// TIA Portal project "FactoryIO_Template_S7-1500_V15_parcial1_terminado" (V15)

(* hardware
DEVICE "S71500/ET200MP-Station_1"  S7-1500 station
   slot 0: "Profilschiene_0"  6ES7 590-1***0-0AA0
   slot 1: "PLC_1"  CPU 1511-1 PN  6ES7 511-1AK00-0AB0  V1.8
   slot 2: "AI 8xU/I/RTD/TC ST_1"  AI 8xU/I/RTD/TC ST  6ES7 531-7KF00-0AB0  V2.0
   slot 3: "AI 8xU/I/RTD/TC ST_2"  AI 8xU/I/RTD/TC ST  6ES7 531-7KF00-0AB0  V2.0
   slot 4: "AI 8xU/I/RTD/TC ST_3"  AI 8xU/I/RTD/TC ST  6ES7 531-7KF00-0AB0  V2.0
   slot 5: "AI 8xU/I/RTD/TC ST_4"  AI 8xU/I/RTD/TC ST  6ES7 531-7KF00-0AB0  V2.0
   slot 6: "DI 16x24VDC BA_1"  DI 16x24VDC BA  6ES7 521-1BH10-0AA0  V1.0
*)

// ===== PLC "PLC_1"  CPU 1511-1 PN =====

VAR_GLOBAL   // PLC tag table "Standard-Variablentabelle"
   "Box_feeder" AT %Q0.0 : Bool;
   "Load_belt" AT %Q0.1 : Bool;
   "Start" AT %I0.0 : Bool;
   "Stop" AT %I0.1 : Bool;
   "Reset" AT %I0.2 : Bool;
   "Manual" AT %I0.3 : Bool;
   "Emergency_stop" AT %I0.5 : Bool;
   "Box_entry" AT %I0.6 : Bool;
   "Turn" AT %Q0.2 : Bool;
   "Pusher_limit" AT %I0.7 : Bool;
   "Push" AT %Q0.3 : Bool;
   "Open_Plate" AT %Q0.4 : Bool;
   "Plate_limit" AT %I1.0 : Bool;
   "Clamp" AT %Q0.5 : Bool;
   "Clamped" AT %I1.1 : Bool;
   "Pallet_feeder" AT %Q0.6 : Bool;
   "Pallet_at_entry" AT %I1.2 : Bool;
   "S1_Elevator_base" AT %I1.3 : Bool;
   "S2_Elevator_base" AT %I1.4 : Bool;
   "Pallet_at_exit" AT %I1.5 : Bool;
   "Exit_conveyor" AT %Q0.7 : Bool;
   "Elevator_moving" AT %I1.6 : Bool;
   "Move_to_limit" AT %Q1.0 : Bool;
   "Elevator_up" AT %Q1.1 : Bool;
   "Warning light" AT %Q1.3 : Bool;
   "Auto" AT %I0.4 : Bool;
   "Elevator_down" AT %Q1.2 : Bool;
   "Contador1" AT %MW10 : Word;
   "Contador2" AT %MW12 : Word;
   "Contador3" AT %MW14 : Word;
   "Contador4" AT %MW16 : Word;
   "Contador5" AT %MW18 : Word;
   "LimiteContador1" AT %MW20 : Word;
   "LimiteContador2" AT %MW22 : Word;
   "Pallet_in_acensor" AT %M100.0 : Bool;
   "Load_pallet" AT %Q1.4 : Bool;
   "Run_machine" AT %M0.0 : Bool;
   "Elevator_Listo_a_cargar" AT %M100.1 : Bool;
   "LimiteContador3" AT %MW24 : Word;
   "Plaforma_llena" AT %M100.2 : Bool;
END_VAR

DATA_BLOCK "GRAPH1_DB"   // DB1
{ S7_Optimized_Access := 'TRUE' }
VERSION : 0.1
// stored: InstanceOfName GRAPH1
"GRAPH1"
BEGIN
END_DATA_BLOCK

DATA_BLOCK "GRAPH2_DB"   // DB2
{ S7_Optimized_Access := 'TRUE' }
VERSION : 0.1
// stored: InstanceOfName GRAPH2
"GRAPH2"
BEGIN
END_DATA_BLOCK

FUNCTION_BLOCK "GRAPH1"   // FB1, GRAPH_PLUS
{ S7_Optimized_Access := 'TRUE' }
VERSION : 0.1
   VAR_INPUT
      OFF_SQ : Bool := false;   // Turn sequence off
      INIT_SQ : Bool := false;   // Set sequence to initial state
      ACK_EF : Bool := false;   // Acknowledge all errors and faults
      S_PREV : Bool := false;   // Output previous step in parameter S_NO
      S_NEXT : Bool := false;   // Indicate next step in parameter S_NO
      SW_AUTO : Bool := false;   // Automatic mode
      SW_TAP : Bool := false;   // Semiautomatic/switch with transition
      SW_TOP : Bool := false;   // Semiautomatic/ignore transition
      SW_MAN : Bool := false;   // Manual mode
      S_SEL : Int := 0;   // Select step to be output to S_NO
      S_ON : Bool := false;   // Activate step indicated in S_NO
      S_OFF : Bool := false;   // Deactivate step indicated S_NO
      T_PUSH : Bool := false;   // Enable transition to switch in semi automatic mode
   END_VAR
   VAR_OUTPUT
      S_NO : Int := 0;   // Step number
      S_MORE : Bool := false;   // More steps are available and can be shown in S_NO
      S_ACTIVE : Bool := false;   // Step indicated in S_NO is active
      ERR_FLT : Bool := false;   // Interlock or supervision group error
      AUTO_ON : Bool := false;   // Automatic mode is active
      TAP_ON : Bool := false;   // Semiautomatic mode/step with transition enabled
      TOP_ON : Bool := false;   // Semiautomatic mode/ignore transition enabled
      MAN_ON : Bool := false;   // Manual mode is active
   END_VAR
   VAR
      HMI_INFO : Array[0..8] of UInt;
      IF_PAR : G7_IfParPlus_V2;
      RT_DATA : G7_RTDataPlus_V2;   // Internal data area
      Trans1 : G7_TransitionPlus_V2;   // Transition structure
      Trans2 : G7_TransitionPlus_V2;   // Transition structure
      Trans3 : G7_TransitionPlus_V2;   // Transition structure
      Trans4 : G7_TransitionPlus_V2;   // Transition structure
      Trans10 : G7_TransitionPlus_V2;   // Transition structure
      Trans12 : G7_TransitionPlus_V2;   // Transition structure
      Trans13 : G7_TransitionPlus_V2;   // Transition structure
      Trans16 : G7_TransitionPlus_V2;   // Transition structure
      Trans17 : G7_TransitionPlus_V2;   // Transition structure
      Trans18 : G7_TransitionPlus_V2;   // Transition structure
      Trans22 : G7_TransitionPlus_V2;   // Transition structure
      Trans24 : G7_TransitionPlus_V2;   // Transition structure
      Trans25 : G7_TransitionPlus_V2;   // Transition structure
      Trans26 : G7_TransitionPlus_V2;   // Transition structure
      Trans27 : G7_TransitionPlus_V2;   // Transition structure
      Trans28 : G7_TransitionPlus_V2;   // Transition structure
      Reposo : G7_StepPlus_V2;   // Step structure
      Bandas_ON : G7_StepPlus_V2;   // Step structure
      Caja_en_psoicion : G7_StepPlus_V2;   // Step structure
      haciendo_push : G7_StepPlus_V2;   // Step structure
      Saliendo_push : G7_StepPlus_V2;   // Step structure
      Push_afuera_regrese : G7_StepPlus_V2;   // Step structure
      Push_regresando : G7_StepPlus_V2;   // Step structure
      box_hacia_load_belt : G7_StepPlus_V2;   // Step structure
      Avanzando_box_en_load_belt : G7_StepPlus_V2;   // Step structure
      Push_en_inicio : G7_StepPlus_V2;   // Step structure
      "6_cajas_en_plato" : G7_StepPlus_V2;   // Step structure
      Intercambiar_sin_turn : G7_StepPlus_V2;   // Step structure
      Intercambiar_con_turn : G7_StepPlus_V2;   // Step structure
      SINI : Array[0..1] of USInt;
      LSTT : Array[0..15] of USInt;
      ATAJ : Array[0..15] of USInt;
      ATAB : Array[0..15] of USInt;
      PSTT : Array[0..15] of USInt;
      NSTT : Array[0..15] of USInt;
      ASSJ : Array[0..12] of USInt;
      ASSB : Array[0..12] of USInt;
      PTTS : Array[0..12] of USInt;
      NTTS : Array[0..12] of USInt;
      SW_SQTS : Array[0..12] of USInt;
      SWITCH : Array[0..4] of USInt;
      TVX : Array[0..7] of USInt;
      TTX : Array[0..7] of USInt;
      TSX : Array[0..1] of USInt;
      S00X : Array[0..1] of USInt;
      SOFFX : Array[0..1] of USInt;
      SONX : Array[0..1] of USInt;
      SAX : Array[0..1] of USInt;
      SERRX : Array[0..13] of USInt;
      SMX : Array[0..13] of USInt;
      S0X : Array[0..13] of USInt;
      S1X : Array[0..13] of USInt;
      IL_ALARM_INST : Program_Alarm;
      SUP_ALARM_INST : Program_Alarm;
      STEP_TIME_ALARM_INST : Program_Alarm;
      IEC_TIMER_INST : IEC_TIMER;
      TRANSACTION_FLAG : Bool := false;
   END_VAR
   // SINI[0] := 2;
   // LSTT[0] := 255;
   // ATAJ[1] := 1;
   // ATAB[1] := 1;
   // PSTT[1] := 1;
   // NSTT[0] := 1;
   // ASSJ[1] := 1;
   // ASSB[1] := 1;
   // PTTS[0] := 255;
   // NTTS[1] := 1;
   // TVX[0] := 16#1;
   // TTX[0] := 16#1;
   // TSX[0] := 16#1;
   // S00X[0] := 16#1;
   // SOFFX[0] := 16#1;
   // SONX[0] := 16#1;
   // SAX[0] := 16#1;
   // SERRX[0] := 16#1;
   // SMX[0] := 16#1;
   // S0X[0] := 16#1;
   // S1X[0] := 16#1;
   // LSTT[1] := 255;
   // LSTT[2] := 255;
   // LSTT[3] := 255;
   // ATAJ[2] := 2;
   // ATAJ[3] := 3;
   // ATAJ[4] := 4;
   // ATAJ[5] := 5;
   // ATAB[2] := 3;
   // ATAB[3] := 2;
   // ATAB[4] := 4;
   // ATAB[5] := 5;
   // PSTT[2] := 2;
   // PSTT[3] := 2;
   // PSTT[4] := 3;
   // PSTT[5] := 4;
   // NSTT[1] := 2;
   // NSTT[2] := 3;
   // NSTT[3] := 7;
   // ASSJ[2] := 2;
   // ASSJ[3] := 3;
   // ASSJ[4] := 4;
   // ASSB[2] := 2;
   // ASSB[3] := 3;
   // ASSB[4] := 4;
   // PTTS[2] := 1;
   // PTTS[3] := 2;
   // PTTS[4] := 4;
   // NTTS[2] := 2;
   // NTTS[3] := 4;
   // NTTS[4] := 5;
   // SW_SQTS[3] := 1;
   // SW_SQTS[4] := 1;
   // LSTT[5] := 255;
   // NSTT[5] := 5;
   // LSTT[4] := 255;
   // LSTT[6] := 255;
   // LSTT[7] := 255;
   // ATAJ[6] := 6;
   // ATAJ[7] := 7;
   // ATAB[6] := 6;
   // ATAB[7] := 7;
   // PSTT[6] := 5;
   // PSTT[7] := 7;
   // NSTT[4] := 4;
   // NSTT[6] := 6;
   // NSTT[7] := 8;
   // ASSJ[5] := 5;
   // ASSJ[6] := 6;
   // ASSB[5] := 5;
   // ASSB[6] := 6;
   // PTTS[5] := 5;
   // PTTS[6] := 6;
   // NTTS[5] := 6;
   // NTTS[6] := 9;
   // SW_SQTS[5] := 1;
   // SW_SQTS[6] := 1;
   // LSTT[8] := 2;
   // LSTT[9] := 255;
   // LSTT[10] := 255;
   // ATAJ[8] := 8;
   // ATAJ[9] := 9;
   // ATAJ[10] := 10;
   // ATAB[8] := 8;
   // ATAB[9] := 9;
   // ATAB[10] := 15;
   // PSTT[8] := 8;
   // PSTT[9] := 6;
   // PSTT[10] := 9;
   // NSTT[8] := 2;
   // NSTT[9] := 9;
   // NSTT[10] := 10;
   // ASSJ[7] := 7;
   // ASSJ[8] := 8;
   // ASSB[7] := 7;
   // ASSB[8] := 8;
   // PTTS[7] := 3;
   // PTTS[8] := 7;
   // NTTS[7] := 7;
   // NTTS[8] := 8;
   // SW_SQTS[7] := 2;
   // SW_SQTS[8] := 2;
   // ATAB[11] := 12;
   // ATAJ[11] := 11;
   // LSTT[11] := 255;
   // PSTT[11] := 10;
   // NSTT[11] := 12;
   // ASSJ[9] := 9;
   // ASSB[9] := 9;
   // PTTS[9] := 9;
   // NTTS[9] := 10;
   // SW_SQTS[9] := 1;
   // LSTT[12] := 255;
   // LSTT[13] := 2;
   // LSTT[14] := 2;
   // LSTT[15] := 2;
   // ATAJ[12] := 12;
   // ATAJ[13] := 13;
   // ATAJ[14] := 14;
   // ATAJ[15] := 15;
   // ATAB[12] := 11;
   // ATAB[13] := 13;
   // ATAB[14] := 14;
   // ATAB[15] := 10;
   // PSTT[12] := 10;
   // PSTT[13] := 11;
   // PSTT[14] := 12;
   // PSTT[15] := 9;
   // NSTT[12] := 11;
   // NSTT[13] := 2;
   // NSTT[14] := 2;
   // NSTT[15] := 2;
   // ASSJ[10] := 10;
   // ASSJ[11] := 11;
   // ASSJ[12] := 12;
   // ASSB[10] := 10;
   // ASSB[11] := 11;
   // ASSB[12] := 12;
   // PTTS[10] := 10;
   // PTTS[11] := 12;
   // PTTS[12] := 11;
   // NTTS[10] := 12;
   // NTTS[11] := 13;
   // NTTS[12] := 14;
   // SW_SQTS[10] := 3;
   // SW_SQTS[11] := 4;
   // SW_SQTS[12] := 5;
BEGIN
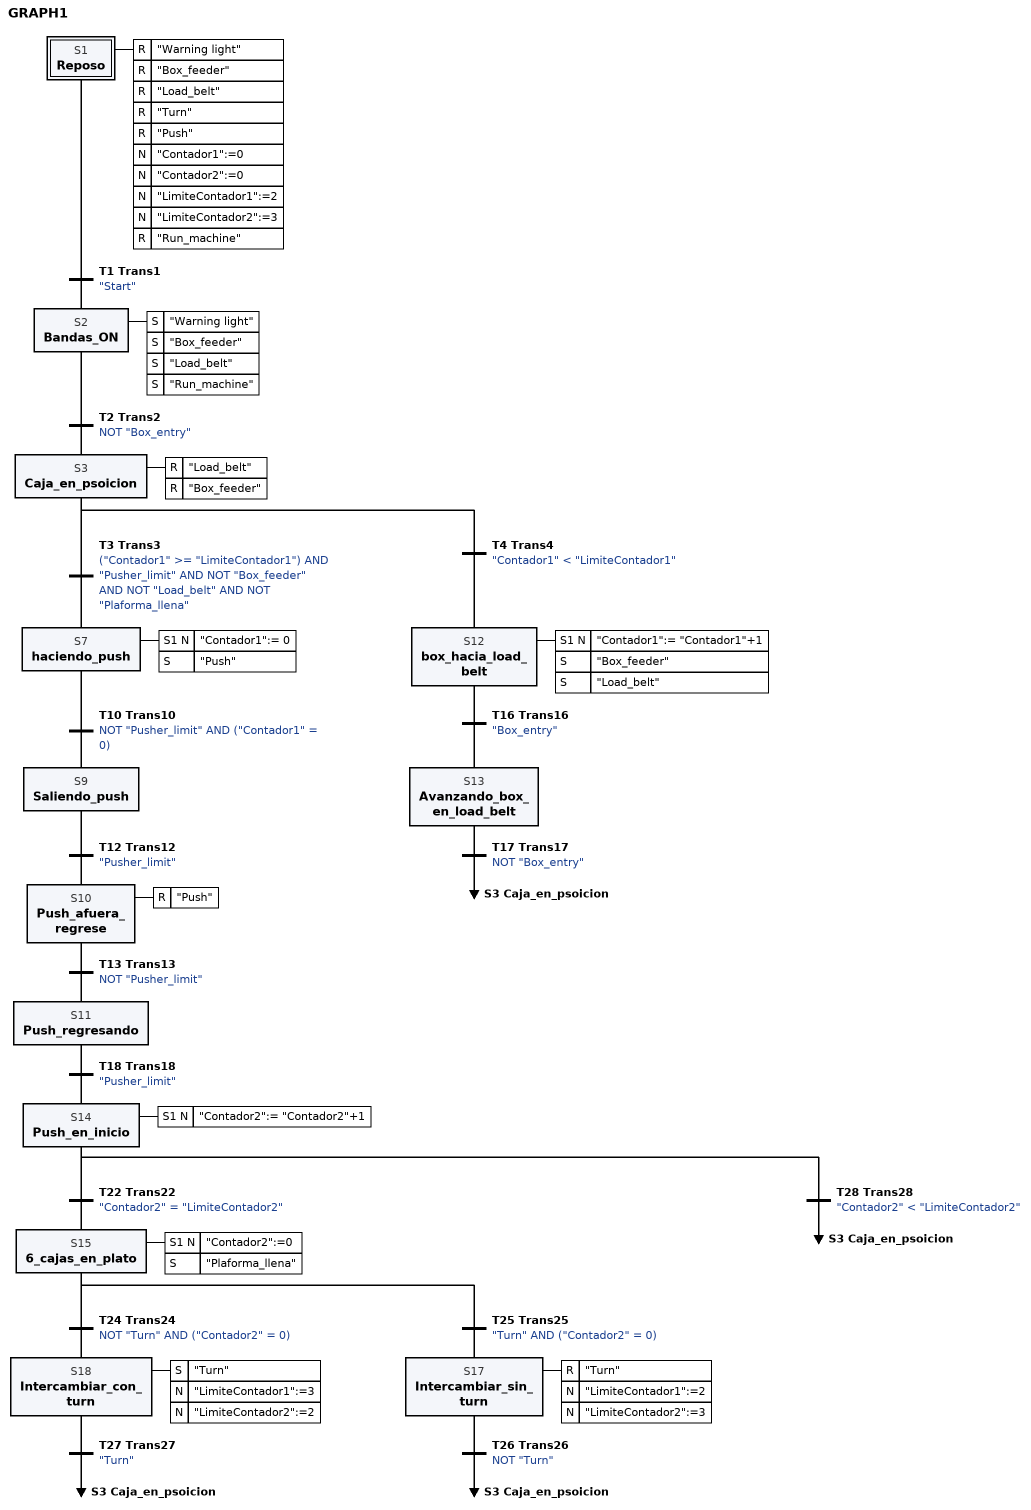
   // sequencer 1
   INITIAL_STEP Reposo:   // S1, max time T#10S, warning time T#7S
              R    "Warning light"
              R    "Box_feeder"
              R    "Load_belt"
              R    "Turn"
              R    "Push"
              N    "Contador1":=0
              N    "Contador2":=0
              N    "LimiteContador1":=2
              N    "LimiteContador2":=3
              R    "Run_machine"
   END_STEP
   TRANSITION Trans1 FROM Reposo TO Bandas_ON   // T1
      := "Start";
   END_TRANSITION
   STEP Bandas_ON:   // S2, max time T#10S, warning time T#7S
              S    "Warning light"
              S    "Box_feeder"
              S    "Load_belt"
              S    "Run_machine"
   END_STEP
   TRANSITION Trans2 FROM Bandas_ON TO Caja_en_psoicion   // T2
      := NOT "Box_entry";
   END_TRANSITION
   STEP Caja_en_psoicion:   // S3, max time T#10S, warning time T#7S
              R    "Load_belt"
              R    "Box_feeder"
   END_STEP
   TRANSITION Trans3 FROM Caja_en_psoicion TO haciendo_push   // T3
      := ("Contador1" >= "LimiteContador1") AND "Pusher_limit" AND NOT "Box_feeder" AND NOT "Load_belt" AND NOT "Plaforma_llena";
   END_TRANSITION
   TRANSITION Trans4 FROM Caja_en_psoicion TO box_hacia_load_belt   // T4
      := "Contador1" < "LimiteContador1";
   END_TRANSITION
   STEP haciendo_push:   // S7, max time T#10S, warning time T#7S
          S1  N    "Contador1":= 0
              S    "Push"
   END_STEP
   TRANSITION Trans10 FROM haciendo_push TO Saliendo_push   // T10
      := NOT "Pusher_limit" AND ("Contador1" = 0);
   END_TRANSITION
   STEP Push_regresando:   // S11, max time T#10S, warning time T#7S
   END_STEP
   TRANSITION Trans18 FROM Push_regresando TO Push_en_inicio   // T18
      := "Pusher_limit";
   END_TRANSITION
   STEP Saliendo_push:   // S9, max time T#10S, warning time T#7S
   END_STEP
   TRANSITION Trans12 FROM Saliendo_push TO Push_afuera_regrese   // T12
      := "Pusher_limit";
   END_TRANSITION
   STEP Push_afuera_regrese:   // S10, max time T#10S, warning time T#7S
              R    "Push"
   END_STEP
   TRANSITION Trans13 FROM Push_afuera_regrese TO Push_regresando   // T13
      := NOT "Pusher_limit";
   END_TRANSITION
   STEP box_hacia_load_belt:   // S12, max time T#10S, warning time T#7S
          S1  N    "Contador1":= "Contador1"+1
              S    "Box_feeder"
              S    "Load_belt"
   END_STEP
   TRANSITION Trans16 FROM box_hacia_load_belt TO Avanzando_box_en_load_belt   // T16
      := "Box_entry";
   END_TRANSITION
   STEP Avanzando_box_en_load_belt:   // S13, max time T#10S, warning time T#7S
   END_STEP
   TRANSITION Trans17 FROM Avanzando_box_en_load_belt TO Caja_en_psoicion   // T17, jump
      := NOT "Box_entry";
   END_TRANSITION
   STEP Push_en_inicio:   // S14, max time T#10S, warning time T#7S
          S1  N    "Contador2":= "Contador2"+1
   END_STEP
   TRANSITION Trans22 FROM Push_en_inicio TO "6_cajas_en_plato"   // T22
      := "Contador2" = "LimiteContador2";
   END_TRANSITION
   TRANSITION Trans28 FROM Push_en_inicio TO Caja_en_psoicion   // T28, jump
      := "Contador2" < "LimiteContador2";
   END_TRANSITION
   STEP "6_cajas_en_plato":   // S15, max time T#10S, warning time T#7S
          S1  N    "Contador2":=0
              S    "Plaforma_llena"
   END_STEP
   TRANSITION Trans24 FROM "6_cajas_en_plato" TO Intercambiar_con_turn   // T24
      := NOT "Turn" AND ("Contador2" = 0);
   END_TRANSITION
   TRANSITION Trans25 FROM "6_cajas_en_plato" TO Intercambiar_sin_turn   // T25
      := "Turn" AND ("Contador2" = 0);
   END_TRANSITION
   STEP Intercambiar_sin_turn:   // S17, max time T#10S, warning time T#7S
              R    "Turn"
              N    "LimiteContador1":=2
              N    "LimiteContador2":=3
   END_STEP
   TRANSITION Trans26 FROM Intercambiar_sin_turn TO Caja_en_psoicion   // T26, jump
      := NOT "Turn";
   END_TRANSITION
   STEP Intercambiar_con_turn:   // S18, max time T#10S, warning time T#7S
              S    "Turn"
              N    "LimiteContador1":=3
              N    "LimiteContador2":=2
   END_STEP
   TRANSITION Trans27 FROM Intercambiar_con_turn TO Caja_en_psoicion   // T27, jump
      := "Turn";
   END_TRANSITION
END_FUNCTION_BLOCK

FUNCTION_BLOCK "GRAPH2"   // FB2, GRAPH_PLUS
{ S7_Optimized_Access := 'TRUE' }
VERSION : 0.1
   VAR_INPUT
      OFF_SQ : Bool := false;   // Turn sequence off
      INIT_SQ : Bool := false;   // Set sequence to initial state
      ACK_EF : Bool := false;   // Acknowledge all errors and faults
      S_PREV : Bool := false;   // Output previous step in parameter S_NO
      S_NEXT : Bool := false;   // Indicate next step in parameter S_NO
      SW_AUTO : Bool := false;   // Automatic mode
      SW_TAP : Bool := false;   // Semiautomatic/switch with transition
      SW_TOP : Bool := false;   // Semiautomatic/ignore transition
      SW_MAN : Bool := false;   // Manual mode
      S_SEL : Int := 0;   // Select step to be output to S_NO
      S_ON : Bool := false;   // Activate step indicated in S_NO
      S_OFF : Bool := false;   // Deactivate step indicated S_NO
      T_PUSH : Bool := false;   // Enable transition to switch in semi automatic mode
   END_VAR
   VAR_OUTPUT
      S_NO : Int := 0;   // Step number
      S_MORE : Bool := false;   // More steps are available and can be shown in S_NO
      S_ACTIVE : Bool := false;   // Step indicated in S_NO is active
      ERR_FLT : Bool := false;   // Interlock or supervision group error
      AUTO_ON : Bool := false;   // Automatic mode is active
      TAP_ON : Bool := false;   // Semiautomatic mode/step with transition enabled
      TOP_ON : Bool := false;   // Semiautomatic mode/ignore transition enabled
      MAN_ON : Bool := false;   // Manual mode is active
   END_VAR
   VAR
      HMI_INFO : Array[0..8] of UInt;
      IF_PAR : G7_IfParPlus_V2;
      RT_DATA : G7_RTDataPlus_V2;   // Internal data area
      Trans1 : G7_TransitionPlus_V2;   // Transition structure
      Trans2 : G7_TransitionPlus_V2;   // Transition structure
      Trans9 : G7_TransitionPlus_V2;   // Transition structure
      Trans10 : G7_TransitionPlus_V2;   // Transition structure
      Trans11 : G7_TransitionPlus_V2;   // Transition structure
      Trans12 : G7_TransitionPlus_V2;   // Transition structure
      Trans14 : G7_TransitionPlus_V2;   // Transition structure
      Trans15 : G7_TransitionPlus_V2;   // Transition structure
      Trans16 : G7_TransitionPlus_V2;   // Transition structure
      Trans17 : G7_TransitionPlus_V2;   // Transition structure
      Trans18 : G7_TransitionPlus_V2;   // Transition structure
      Trans19 : G7_TransitionPlus_V2;   // Transition structure
      Trans20 : G7_TransitionPlus_V2;   // Transition structure
      Trans21 : G7_TransitionPlus_V2;   // Transition structure
      Trans22 : G7_TransitionPlus_V2;   // Transition structure
      Trans23 : G7_TransitionPlus_V2;   // Transition structure
      Trans24 : G7_TransitionPlus_V2;   // Transition structure
      Trans25 : G7_TransitionPlus_V2;   // Transition structure
      Trans27 : G7_TransitionPlus_V2;   // Transition structure
      Trans28 : G7_TransitionPlus_V2;   // Transition structure
      Trans29 : G7_TransitionPlus_V2;   // Transition structure
      Trans30 : G7_TransitionPlus_V2;   // Transition structure
      Trans31 : G7_TransitionPlus_V2;   // Transition structure
      Trans32 : G7_TransitionPlus_V2;   // Transition structure
      Trans33 : G7_TransitionPlus_V2;   // Transition structure
      Reposo_inferior : G7_StepPlus_V2;   // Step structure
      Pallet_avanzando : G7_StepPlus_V2;   // Step structure
      Pallet_en_posicion : G7_StepPlus_V2;   // Step structure
      Entrando_a_load_pallet : G7_StepPlus_V2;   // Step structure
      Muevo_ascensor : G7_StepPlus_V2;   // Step structure
      Acomodar_pallet : G7_StepPlus_V2;   // Step structure
      Step11 : G7_StepPlus_V2;   // Step structure
      acesor_subiendo : G7_StepPlus_V2;   // Step structure
      elevator_arriba : G7_StepPlus_V2;   // Step structure
      Empezar_descarga_activar_clamp : G7_StepPlus_V2;   // Step structure
      cajas_sujetas_a_descargar : G7_StepPlus_V2;   // Step structure
      plate_abriendo : G7_StepPlus_V2;   // Step structure
      plate_abierto : G7_StepPlus_V2;   // Step structure
      Cajas_en_pallet : G7_StepPlus_V2;   // Step structure
      elvator_bajando : G7_StepPlus_V2;   // Step structure
      elvator_bajo_1 : G7_StepPlus_V2;   // Step structure
      Cerrando_plato : G7_StepPlus_V2;   // Step structure
      plato_cerrado : G7_StepPlus_V2;   // Step structure
      Elevador_lleno : G7_StepPlus_V2;   // Step structure
      Acensor_bajando : G7_StepPlus_V2;   // Step structure
      Asensor_abajo : G7_StepPlus_V2;   // Step structure
      Pallet_Saliendo_de_elevador : G7_StepPlus_V2;   // Step structure
      Step27 : G7_StepPlus_V2;   // Step structure
      SINI : Array[0..1] of USInt;
      LSTT : Array[0..24] of USInt;
      ATAJ : Array[0..24] of USInt;
      ATAB : Array[0..24] of USInt;
      PSTT : Array[0..24] of USInt;
      NSTT : Array[0..24] of USInt;
      ASSJ : Array[0..22] of USInt;
      ASSB : Array[0..22] of USInt;
      PTTS : Array[0..22] of USInt;
      NTTS : Array[0..22] of USInt;
      SW_SQTS : Array[0..22] of USInt;
      SWITCH : Array[0..1] of USInt;
      TVX : Array[0..5] of USInt;
      TTX : Array[0..5] of USInt;
      TSX : Array[0..1] of USInt;
      S00X : Array[0..1] of USInt;
      SOFFX : Array[0..1] of USInt;
      SONX : Array[0..1] of USInt;
      SAX : Array[0..1] of USInt;
      SERRX : Array[0..23] of USInt;
      SMX : Array[0..23] of USInt;
      S0X : Array[0..23] of USInt;
      S1X : Array[0..23] of USInt;
      IL_ALARM_INST : Program_Alarm;
      SUP_ALARM_INST : Program_Alarm;
      STEP_TIME_ALARM_INST : Program_Alarm;
      IEC_TIMER_INST : IEC_TIMER;
      TRANSACTION_FLAG : Bool := false;
   END_VAR
   // SINI[0] := 2;
   // LSTT[0] := 255;
   // LSTT[1] := 255;
   // LSTT[2] := 255;
   // LSTT[3] := 255;
   // ATAJ[1] := 1;
   // ATAJ[2] := 2;
   // ATAJ[3] := 3;
   // ATAB[1] := 1;
   // ATAB[2] := 2;
   // ATAB[3] := 4;
   // PSTT[1] := 1;
   // PSTT[2] := 3;
   // PSTT[3] := 2;
   // NSTT[0] := 1;
   // NSTT[1] := 3;
   // NSTT[2] := 2;
   // NSTT[3] := 5;
   // ASSJ[1] := 1;
   // ASSJ[2] := 2;
   // ASSJ[3] := 3;
   // ASSB[1] := 1;
   // ASSB[2] := 2;
   // ASSB[3] := 3;
   // PTTS[0] := 255;
   // PTTS[2] := 2;
   // PTTS[3] := 1;
   // NTTS[1] := 1;
   // NTTS[2] := 4;
   // NTTS[3] := 2;
   // TVX[0] := 16#1;
   // TTX[0] := 16#1;
   // TSX[0] := 16#1;
   // S00X[0] := 16#1;
   // SOFFX[0] := 16#1;
   // SONX[0] := 16#1;
   // SAX[0] := 16#1;
   // SERRX[0] := 16#1;
   // SMX[0] := 16#1;
   // S0X[0] := 16#1;
   // S1X[0] := 16#1;
   // LSTT[4] := 255;
   // LSTT[5] := 255;
   // LSTT[6] := 2;
   // LSTT[7] := 255;
   // ATAJ[4] := 4;
   // ATAJ[5] := 5;
   // ATAJ[6] := 6;
   // ATAJ[7] := 7;
   // ATAB[4] := 3;
   // ATAB[5] := 5;
   // ATAB[6] := 6;
   // ATAB[7] := 7;
   // PSTT[4] := 2;
   // PSTT[5] := 5;
   // PSTT[6] := 6;
   // PSTT[7] := 4;
   // NSTT[4] := 4;
   // NSTT[5] := 6;
   // NSTT[6] := 2;
   // NSTT[7] := 7;
   // ASSJ[4] := 4;
   // ASSJ[5] := 5;
   // ASSJ[6] := 6;
   // ASSB[4] := 4;
   // ASSB[5] := 5;
   // ASSB[6] := 6;
   // PTTS[4] := 4;
   // PTTS[5] := 3;
   // PTTS[6] := 5;
   // NTTS[4] := 7;
   // NTTS[5] := 5;
   // NTTS[6] := 6;
   // SW_SQTS[4] := 1;
   // SW_SQTS[5] := 2;
   // SW_SQTS[6] := 2;
   // LSTT[8] := 255;
   // LSTT[9] := 255;
   // ATAJ[8] := 8;
   // ATAJ[9] := 9;
   // ATAB[8] := 8;
   // ATAB[9] := 9;
   // PSTT[8] := 7;
   // PSTT[9] := 8;
   // NSTT[8] := 8;
   // NSTT[9] := 9;
   // ASSJ[7] := 7;
   // ASSJ[8] := 8;
   // ASSB[7] := 7;
   // ASSB[8] := 8;
   // PTTS[7] := 7;
   // PTTS[8] := 8;
   // NTTS[7] := 8;
   // NTTS[8] := 9;
   // SW_SQTS[7] := 1;
   // SW_SQTS[8] := 1;
   // LSTT[10] := 255;
   // LSTT[11] := 255;
   // LSTT[12] := 255;
   // LSTT[13] := 255;
   // LSTT[14] := 255;
   // LSTT[15] := 255;
   // LSTT[16] := 255;
   // LSTT[17] := 255;
   // LSTT[18] := 255;
   // ATAJ[10] := 10;
   // ATAJ[11] := 11;
   // ATAJ[12] := 12;
   // ATAJ[13] := 13;
   // ATAJ[14] := 14;
   // ATAJ[15] := 15;
   // ATAJ[16] := 16;
   // ATAJ[17] := 17;
   // ATAJ[18] := 18;
   // ATAB[10] := 10;
   // ATAB[11] := 11;
   // ATAB[12] := 12;
   // ATAB[13] := 13;
   // ATAB[14] := 14;
   // ATAB[15] := 15;
   // ATAB[16] := 16;
   // ATAB[17] := 17;
   // ATAB[18] := 19;
   // PSTT[10] := 9;
   // PSTT[11] := 10;
   // PSTT[12] := 11;
   // PSTT[13] := 12;
   // PSTT[14] := 13;
   // PSTT[15] := 14;
   // PSTT[16] := 15;
   // PSTT[17] := 16;
   // PSTT[18] := 17;
   // NSTT[10] := 10;
   // NSTT[11] := 11;
   // NSTT[12] := 12;
   // NSTT[13] := 13;
   // NSTT[14] := 14;
   // NSTT[15] := 15;
   // NSTT[16] := 16;
   // NSTT[17] := 17;
   // NSTT[18] := 18;
   // ASSJ[9] := 9;
   // ASSJ[10] := 10;
   // ASSJ[11] := 11;
   // ASSJ[12] := 12;
   // ASSJ[13] := 13;
   // ASSJ[14] := 14;
   // ASSJ[15] := 15;
   // ASSJ[16] := 16;
   // ASSJ[17] := 17;
   // ASSB[9] := 9;
   // ASSB[10] := 10;
   // ASSB[11] := 11;
   // ASSB[12] := 12;
   // ASSB[13] := 13;
   // ASSB[14] := 14;
   // ASSB[15] := 15;
   // ASSB[16] := 16;
   // ASSB[17] := 17;
   // PTTS[9] := 9;
   // PTTS[10] := 10;
   // PTTS[11] := 11;
   // PTTS[12] := 12;
   // PTTS[13] := 13;
   // PTTS[14] := 14;
   // PTTS[15] := 15;
   // PTTS[16] := 16;
   // PTTS[17] := 17;
   // NTTS[9] := 10;
   // NTTS[10] := 11;
   // NTTS[11] := 12;
   // NTTS[12] := 13;
   // NTTS[13] := 14;
   // NTTS[14] := 15;
   // NTTS[15] := 16;
   // NTTS[16] := 17;
   // NTTS[17] := 18;
   // SW_SQTS[9] := 1;
   // SW_SQTS[10] := 1;
   // SW_SQTS[11] := 1;
   // SW_SQTS[12] := 1;
   // SW_SQTS[13] := 1;
   // SW_SQTS[14] := 1;
   // SW_SQTS[15] := 1;
   // SW_SQTS[16] := 1;
   // SW_SQTS[17] := 1;
   // LSTT[19] := 8;
   // LSTT[20] := 255;
   // ATAJ[19] := 19;
   // ATAJ[20] := 20;
   // ATAB[19] := 18;
   // ATAB[20] := 20;
   // PSTT[19] := 17;
   // PSTT[20] := 18;
   // NSTT[19] := 8;
   // NSTT[20] := 19;
   // ASSJ[18] := 18;
   // ASSB[18] := 18;
   // PTTS[18] := 18;
   // NTTS[18] := 20;
   // SW_SQTS[18] := 3;
   // LSTT[21] := 255;
   // LSTT[22] := 255;
   // LSTT[23] := 255;
   // LSTT[24] := 1;
   // ATAJ[21] := 21;
   // ATAJ[22] := 22;
   // ATAJ[23] := 23;
   // ATAJ[24] := 24;
   // ATAB[21] := 21;
   // ATAB[22] := 22;
   // ATAB[23] := 23;
   // ATAB[24] := 24;
   // PSTT[21] := 19;
   // PSTT[22] := 20;
   // PSTT[23] := 21;
   // PSTT[24] := 22;
   // NSTT[21] := 20;
   // NSTT[22] := 21;
   // NSTT[23] := 22;
   // NSTT[24] := 1;
   // ASSJ[19] := 19;
   // ASSJ[20] := 20;
   // ASSJ[21] := 21;
   // ASSJ[22] := 22;
   // ASSB[19] := 19;
   // ASSB[20] := 20;
   // ASSB[21] := 21;
   // ASSB[22] := 22;
   // PTTS[19] := 20;
   // PTTS[20] := 21;
   // PTTS[21] := 22;
   // PTTS[22] := 23;
   // NTTS[19] := 21;
   // NTTS[20] := 22;
   // NTTS[21] := 23;
   // NTTS[22] := 24;
   // SW_SQTS[19] := 3;
   // SW_SQTS[20] := 3;
   // SW_SQTS[21] := 3;
   // SW_SQTS[22] := 3;
BEGIN
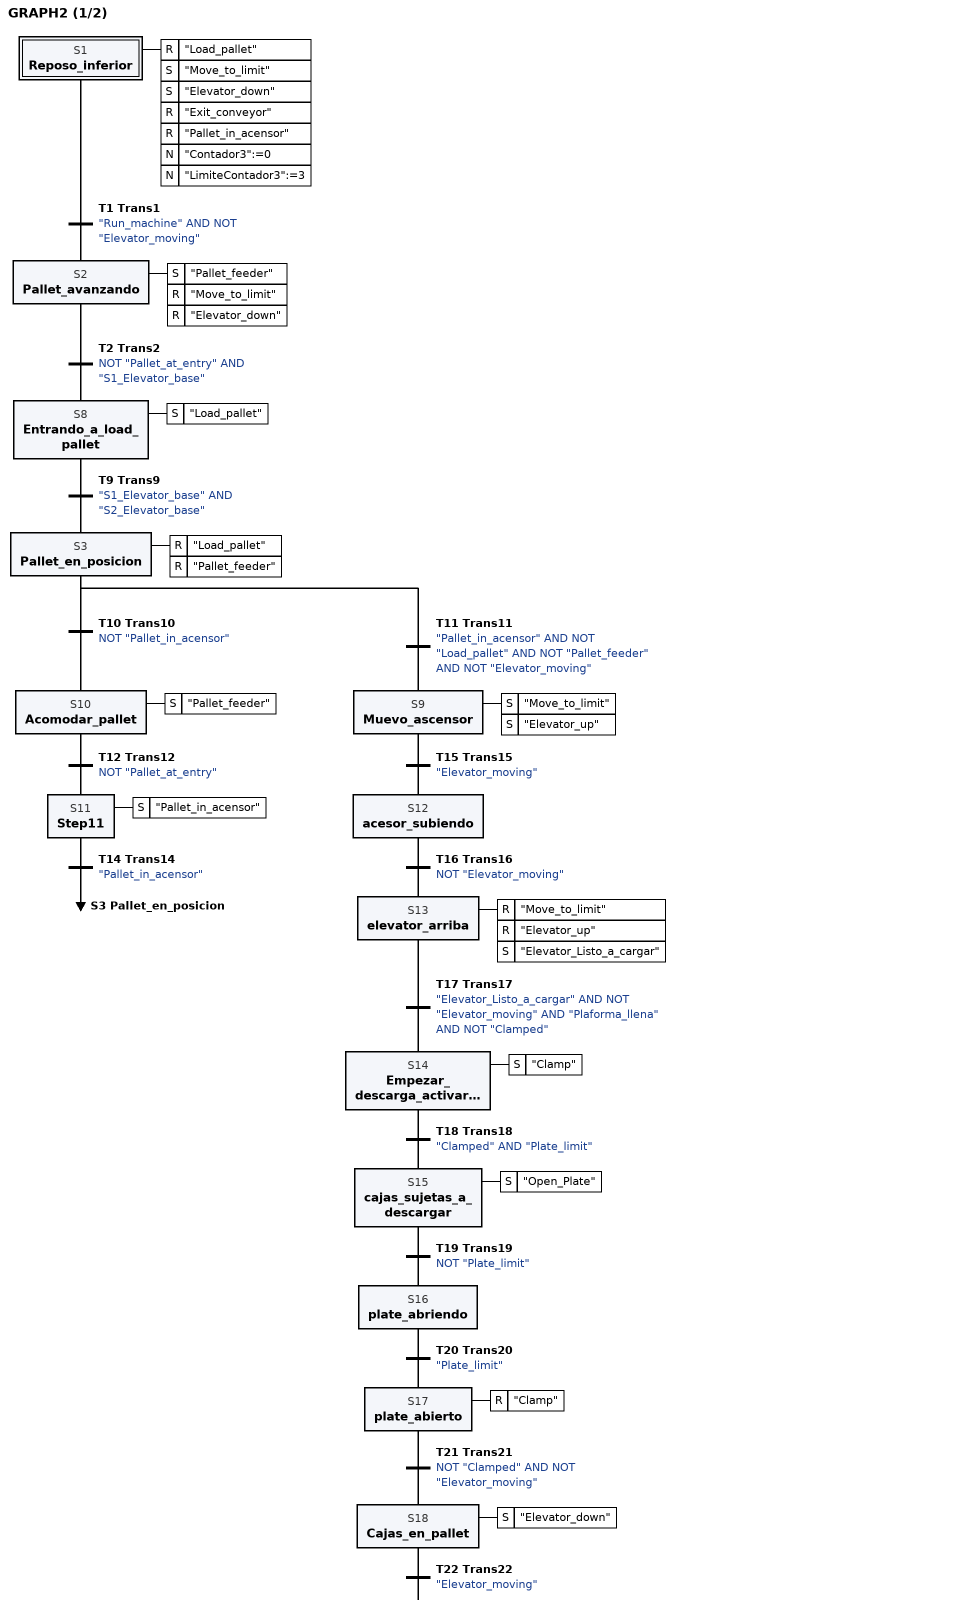
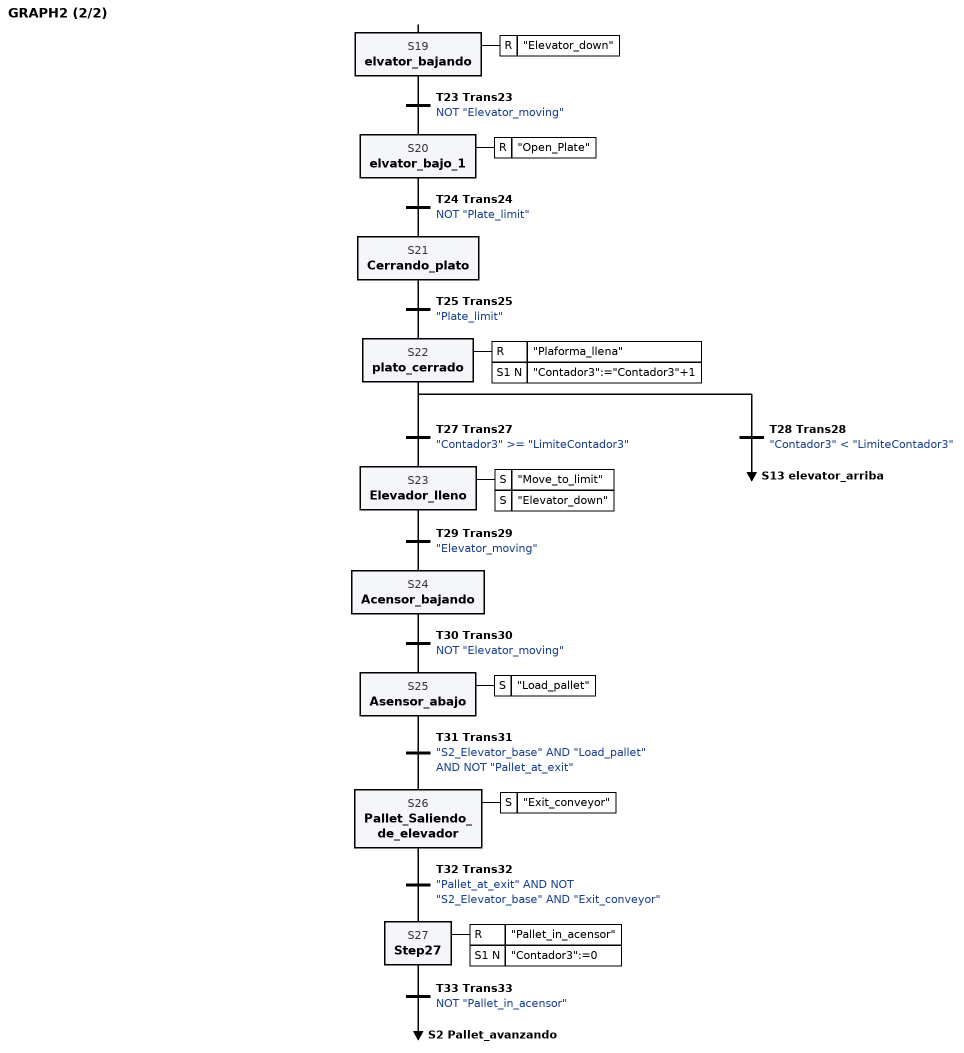
   // sequencer 1
   INITIAL_STEP Reposo_inferior:   // S1, max time T#10S, warning time T#7S
              R    "Load_pallet"
              S    "Move_to_limit"
              S    "Elevator_down"
              R    "Exit_conveyor"
              R    "Pallet_in_acensor"
              N    "Contador3":=0
              N    "LimiteContador3":=3
   END_STEP
   TRANSITION Trans1 FROM Reposo_inferior TO Pallet_avanzando   // T1
      := "Run_machine" AND NOT "Elevator_moving";
   END_TRANSITION
   STEP Pallet_avanzando:   // S2, max time T#10S, warning time T#7S
              S    "Pallet_feeder"
              R    "Move_to_limit"
              R    "Elevator_down"
   END_STEP
   TRANSITION Trans2 FROM Pallet_avanzando TO Entrando_a_load_pallet   // T2
      := NOT "Pallet_at_entry" AND "S1_Elevator_base";
   END_TRANSITION
   STEP Pallet_en_posicion:   // S3, max time T#10S, warning time T#7S
              R    "Load_pallet"
              R    "Pallet_feeder"
   END_STEP
   TRANSITION Trans10 FROM Pallet_en_posicion TO Acomodar_pallet   // T10
      := NOT "Pallet_in_acensor";
   END_TRANSITION
   TRANSITION Trans11 FROM Pallet_en_posicion TO Muevo_ascensor   // T11
      := "Pallet_in_acensor" AND NOT "Load_pallet" AND NOT "Pallet_feeder" AND NOT "Elevator_moving";
   END_TRANSITION
   STEP Muevo_ascensor:   // S9, max time T#10S, warning time T#7S
              S    "Move_to_limit"
              S    "Elevator_up"
   END_STEP
   TRANSITION Trans15 FROM Muevo_ascensor TO acesor_subiendo   // T15
      := "Elevator_moving";
   END_TRANSITION
   STEP Entrando_a_load_pallet:   // S8, max time T#10S, warning time T#7S
              S    "Load_pallet"
   END_STEP
   TRANSITION Trans9 FROM Entrando_a_load_pallet TO Pallet_en_posicion   // T9
      := "S1_Elevator_base" AND "S2_Elevator_base";
   END_TRANSITION
   STEP Acomodar_pallet:   // S10, max time T#10S, warning time T#7S
              S    "Pallet_feeder"
   END_STEP
   TRANSITION Trans12 FROM Acomodar_pallet TO Step11   // T12
      := NOT "Pallet_at_entry";
   END_TRANSITION
   STEP Step11:   // S11, max time T#10S, warning time T#7S
              S    "Pallet_in_acensor"
   END_STEP
   TRANSITION Trans14 FROM Step11 TO Pallet_en_posicion   // T14, jump
      := "Pallet_in_acensor";
   END_TRANSITION
   STEP acesor_subiendo:   // S12, max time T#10S, warning time T#7S
   END_STEP
   TRANSITION Trans16 FROM acesor_subiendo TO elevator_arriba   // T16
      := NOT "Elevator_moving";
   END_TRANSITION
   STEP elevator_arriba:   // S13, max time T#10S, warning time T#7S
              R    "Move_to_limit"
              R    "Elevator_up"
              S    "Elevator_Listo_a_cargar"
   END_STEP
   TRANSITION Trans17 FROM elevator_arriba TO Empezar_descarga_activar_clamp   // T17
      := "Elevator_Listo_a_cargar" AND NOT "Elevator_moving" AND "Plaforma_llena" AND NOT "Clamped";
   END_TRANSITION
   STEP Empezar_descarga_activar_clamp:   // S14, max time T#10S, warning time T#7S
              S    "Clamp"
   END_STEP
   TRANSITION Trans18 FROM Empezar_descarga_activar_clamp TO cajas_sujetas_a_descargar   // T18
      := "Clamped" AND "Plate_limit";
   END_TRANSITION
   STEP cajas_sujetas_a_descargar:   // S15, max time T#10S, warning time T#7S
              S    "Open_Plate"
   END_STEP
   TRANSITION Trans19 FROM cajas_sujetas_a_descargar TO plate_abriendo   // T19
      := NOT "Plate_limit";
   END_TRANSITION
   STEP plate_abriendo:   // S16, max time T#10S, warning time T#7S
   END_STEP
   TRANSITION Trans20 FROM plate_abriendo TO plate_abierto   // T20
      := "Plate_limit";
   END_TRANSITION
   STEP plate_abierto:   // S17, max time T#10S, warning time T#7S
              R    "Clamp"
   END_STEP
   TRANSITION Trans21 FROM plate_abierto TO Cajas_en_pallet   // T21
      := NOT "Clamped" AND NOT "Elevator_moving";
   END_TRANSITION
   STEP Cajas_en_pallet:   // S18, max time T#10S, warning time T#7S
              S    "Elevator_down"
   END_STEP
   TRANSITION Trans22 FROM Cajas_en_pallet TO elvator_bajando   // T22
      := "Elevator_moving";
   END_TRANSITION
   STEP elvator_bajando:   // S19, max time T#10S, warning time T#7S
              R    "Elevator_down"
   END_STEP
   TRANSITION Trans23 FROM elvator_bajando TO elvator_bajo_1   // T23
      := NOT "Elevator_moving";
   END_TRANSITION
   STEP elvator_bajo_1:   // S20, max time T#10S, warning time T#7S
              R    "Open_Plate"
   END_STEP
   TRANSITION Trans24 FROM elvator_bajo_1 TO Cerrando_plato   // T24
      := NOT "Plate_limit";
   END_TRANSITION
   STEP Cerrando_plato:   // S21, max time T#10S, warning time T#7S
   END_STEP
   TRANSITION Trans25 FROM Cerrando_plato TO plato_cerrado   // T25
      := "Plate_limit";
   END_TRANSITION
   STEP plato_cerrado:   // S22, max time T#10S, warning time T#7S
              R    "Plaforma_llena"
          S1  N    "Contador3":="Contador3"+1
   END_STEP
   TRANSITION Trans27 FROM plato_cerrado TO Elevador_lleno   // T27
      := "Contador3" >= "LimiteContador3";
   END_TRANSITION
   TRANSITION Trans28 FROM plato_cerrado TO elevator_arriba   // T28, jump
      := "Contador3" < "LimiteContador3";
   END_TRANSITION
   STEP Elevador_lleno:   // S23, max time T#10S, warning time T#7S
              S    "Move_to_limit"
              S    "Elevator_down"
   END_STEP
   TRANSITION Trans29 FROM Elevador_lleno TO Acensor_bajando   // T29
      := "Elevator_moving";
   END_TRANSITION
   STEP Acensor_bajando:   // S24, max time T#10S, warning time T#7S
   END_STEP
   TRANSITION Trans30 FROM Acensor_bajando TO Asensor_abajo   // T30
      := NOT "Elevator_moving";
   END_TRANSITION
   STEP Asensor_abajo:   // S25, max time T#10S, warning time T#7S
              S    "Load_pallet"
   END_STEP
   TRANSITION Trans31 FROM Asensor_abajo TO Pallet_Saliendo_de_elevador   // T31
      := "S2_Elevator_base" AND "Load_pallet" AND NOT "Pallet_at_exit";
   END_TRANSITION
   STEP Pallet_Saliendo_de_elevador:   // S26, max time T#10S, warning time T#7S
              S    "Exit_conveyor"
   END_STEP
   TRANSITION Trans32 FROM Pallet_Saliendo_de_elevador TO Step27   // T32
      := "Pallet_at_exit" AND NOT "S2_Elevator_base" AND "Exit_conveyor";
   END_TRANSITION
   STEP Step27:   // S27, max time T#10S, warning time T#7S
              R    "Pallet_in_acensor"
          S1  N    "Contador3":=0
   END_STEP
   TRANSITION Trans33 FROM Step27 TO Pallet_avanzando   // T33, jump
      := NOT "Pallet_in_acensor";
   END_TRANSITION
END_FUNCTION_BLOCK

FUNCTION "MHJ-PLC-Lab-Function-S71500" : Void   // FC9000, SCL
{ S7_Optimized_Access := 'TRUE' }
VERSION : 0.1
   VAR_TEMP
      Value : Byte;
      ForCounter : Int;
   END_VAR
   VAR CONSTANT
      Value_01_DW : DWord := 16#1223_5486;
      Value_02_DW : DWord := 16#A6C9_D1F5;
   END_VAR
BEGIN

   #Value:=PEEK(area := 16#82,
        dbNumber := 0,
        byteOffset := 511);
   #Value := #Value + 1;

   POKE(area := 16#82,
        dbNumber := 0,
        byteOffset := 511,
        value := #Value);

   POKE(area := 16#82,
        dbNumber := 0,
        byteOffset := 1016,
        value := #Value_01_DW);
   POKE(area := 16#82,
        dbNumber := 0,
        byteOffset := 1020,
        value := #Value_02_DW);

   FOR #ForCounter := 0 TO 63 DO
       #Value:=PEEK(area := 16#1,
            dbNumber := 0,
            byteOffset := #ForCounter);
       POKE(area := 16#81,
            dbNumber := 0,
            byteOffset := #ForCounter,
            value := #Value);
   END_FOR;
   #Value := PEEK(area := 16#1,
                  dbNumber := 0,
                  byteOffset := 512);
   POKE(area := 16#82,
        dbNumber := 0,
        byteOffset := 512,
        value := #Value);
END_FUNCTION

ORGANIZATION_BLOCK "Main"   // OB1, LAD, ProgramCycle
TITLE = "Main Program Sweep (Cycle)"
{ S7_Optimized_Access := 'TRUE' }
VERSION : 0.1
   VAR_INPUT
      Initial_Call : Bool;   // Initial call of this OB
      Remanence : Bool;   // =True, if remanent data are available
   END_VAR
BEGIN

REGION Network 1
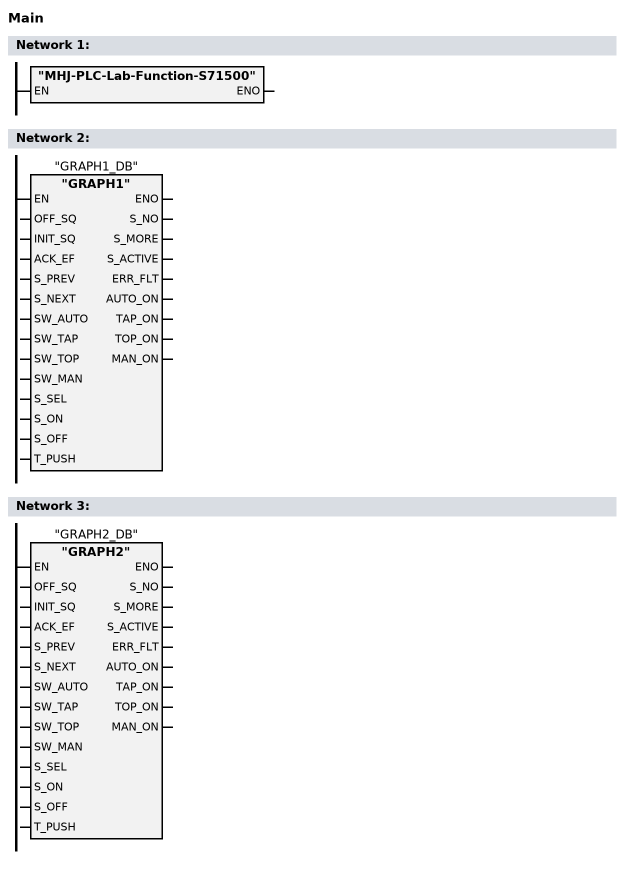
   RUNG wire#powerrail
      "MHJ-PLC-Lab-Function-S71500"()
   END_RUNG
   // the same network as SCL:
   "MHJ-PLC-Lab-Function-S71500"();
END_REGION

REGION Network 2
   RUNG wire#powerrail
      "GRAPH1_DB"(OFF_SQ :=, INIT_SQ :=, ACK_EF :=, S_PREV :=, S_NEXT :=, SW_AUTO :=, SW_TAP :=, SW_TOP :=, SW_MAN :=, S_SEL :=, S_ON :=, S_OFF :=, T_PUSH :=, S_NO =>, S_MORE =>, S_ACTIVE =>, ERR_FLT =>, AUTO_ON =>, TAP_ON =>, TOP_ON =>, MAN_ON =>)
   END_RUNG
   // the same network as SCL:
   "GRAPH1_DB"();   // "GRAPH1"
END_REGION

REGION Network 3
   RUNG wire#powerrail
      "GRAPH2_DB"(OFF_SQ :=, INIT_SQ :=, ACK_EF :=, S_PREV :=, S_NEXT :=, SW_AUTO :=, SW_TAP :=, SW_TOP :=, SW_MAN :=, S_SEL :=, S_ON :=, S_OFF :=, T_PUSH :=, S_NO =>, S_MORE =>, S_ACTIVE =>, ERR_FLT =>, AUTO_ON =>, TAP_ON =>, TOP_ON =>, MAN_ON =>)
   END_RUNG
   // the same network as SCL:
   "GRAPH2_DB"();   // "GRAPH2"
END_REGION
END_ORGANIZATION_BLOCK